{attribute addProperty BoxType "EK1122-0000-0018"}
{attribute addProperty Id "A_0060_AT2020_0250_0019_AT2020_0250A_0060_AT2020_0250_0019_AT2020_0250_D1D8CBA264080Beckhoff_AT2xxxsub_EK1100EK1100_179A0949162A_0001_AT2000_0233_0022AT2000_050BA88864080A_0002_AT2000_0233_0023AT2000_050BA88864080A_0003_AT2000_0233_0024AT2000_050BA88864080A_0004_AT2000_0250_0016AT2000_9506A48267284A_0005_AT2000_0250_0017AT2000_9506A48267284A_0006_AT2000_0250_0018AT2000_9506A48267284A_0007_AT2000_0250_0019AT2000_9506A48267284A_0008_AT2000_0250_0020AT2000_9506A48267284A_0009_AT2000_0250_0021AT2000_9506A48267284A_0010_AT2000_0250_0022AT2000_9506A48267284A_0011_AT2000_0250_0023AT2000_9506A48267284A_0012_AT2001_0250_0016AT2001_9506A48267284A_0013_AT2001_0250_0017AT2001_9506A48267284A_0014_AT2001_0250_0018AT2001_9506A48267284A_0015_AT2001_0250_0019AT2001_9506A48267284A_0016_AT2001_0250_0020AT2001_9506A48267284A_0017_AT2001_0250_0022AT2001_9506A48267284A_0018_AT2001_0250_0023AT2001_9506A48267284A_0019_AT2001_0250_0024AT2001_9506A48267284A_0020_AT2002_0249_0021AT2002_9506A48267284A_0021_AT2002_0249_0022AT2002_9506A48267284A_0022_AT2002_0249_0023AT2002_9506A48267284A_0023_AT2002_0250_0022AT2002_9506A48267284A_0024_AT2002_0250_0023AT2002_9506A48267284A_0025_AT2002_0250_0024AT2002_9506A48267284A_0026_AT2020_0250_0018AT2020_9506A48267284A_0027_AT2020_0250_0021AT2020_9506A48267284A_0028_AT2021_0250_0018AT2021_9506A48267284A_0029_AT2021_0250_0020AT2021_9506A48267284A_0030_AT2025_0250_0018AT2025_9506A48267284A_0031_AT2026_0250_0021AT2026_9506A48267284A_0032_AT2026_0250_0023AT2026_9506A48267284A_0033_AT2040_0250_0018AT2040_9506A48267284A_0034_AT2040_0250_0019AT2040_9506A48267284A_0035_AT2040_0250_0020AT2040_9506A48267284A_0036_AT2040_0250_0021A_0036_AT2040_0250_0021_02D2816B64080A_0037_AT2040_0250_0022A_0037_AT2040_0250_0022_F543FD7364080A_0038_AT2040_0250_0023A_0038_AT2040_0250_0023_F11EC84664080A_0039_AT2040_0250_0024A_0039_AT2040_0250_0024_E1E41A1064080A_0040_AT2041_0250_0018A_0040_AT2041_0250_0018_12B9905D64080A_0041_AT2041_0250_0019A_0041_AT2041_0250_0019_5F65D83164080A_0042_AT2041_0250_0020A_0042_AT2041_0250_0020_102CD79B64080A_0043_AT2041_0250_0021A_0043_AT2041_0250_0021_00D605CD64080A_0044_AT2041_0250_0022A_0044_AT2041_0250_0022_EDE0E1B464080A_0045_AT2041_0250_0023A_0045_AT2041_0250_0023_3AEB85C764080A_0046_AT2042_0250_0024A_0046_AT2042_0250_0024_1AE974B864080A_0047_AT2050_0500_0016A_0047_AT2050_0500_0016_ED7808A064080A_0048_AT2050_0500_0017A_0048_AT2050_0500_0017_6811D0ED64080A_0049_AT2050_0500_0018A_0049_AT2050_0500_0018_289538B264080A_0050_AT2050_0500_0019A_0050_AT2050_0500_0019_16FCA7F964080A_0051_AT2050_0500_0020A_0051_AT2050_0500_0020_887F94A764080A_0052_AT2050_0500_0021A_0052_AT2050_0500_0021_B6160BEC64080A_0053_AT2050_0500_0022A_0053_AT2050_0500_0022_1DEC9EBC64080A_0054_AT2050_0500_0023A_0054_AT2050_0500_0023_99CF05DF64080A_0055_AT2050_0500_0024A_0055_AT2050_0500_0024_061BAB1564080A_0056_AT2050_0501_0017A_0056_AT2050_0501_0017_8372735864080A_0057_AT2050_0501_0020A_0057_AT2050_0501_0020_74E30F4064080A_0058_AT2050_0501_0021A_0058_AT2050_0501_0021_C12219F464080A_0061_AT2020_0250_0023_AT2020_0250A_0061_AT2020_0250_0023_AT2020_0250_98D9E94964080A_0062_AT2025_0250_0020_AT2025_0250A_0062_AT2025_0250_0020_AT2025_0250_D505A12564080A_0063_AT2025_0250_0022_AT2025_0250A_0063_AT2025_0250_0022_AT2025_0250_FB2CCE7664080A_0064_AT2025_0250_0023_AT2025_0250A_0064_AT2025_0250_0023_AT2025_0250_28C9970A64080A_0065_AT2026_0250_0019_AT2026_0250A_0065_AT2026_0250_0019_AT2026_0250_ADA04F4764080A_0066_AT2026_0250_0020_AT2026_0250A_0066_AT2026_0250_0020_AT2026_0250_5A31335F64080A_0067_AT2026_0250_0022_AT2026_0250A_0067_AT2026_0250_0022_AT2026_0250_D8AB0CE364080A_0068_AT2026_0250_0024_AT2026_0250A_0068_AT2026_0250_0024_AT2026_0250_C0DF91BF64080A_0069_AT2050_0501_0019_AT2050_0501A_0069_AT2050_0501_0019_AT2050_0501_33653EE264080A_0070_AT2050_0501_0022_AT2050_0501A_0070_AT2050_0501_0022_AT2050_0501_239FECB464080A_0071_AT2050_0501_0023_AT2050_0501A_0071_AT2050_0501_0023_AT2050_0501_196D5B8364080A_0072_AT2050_0501_0024_AT2050_0501A_0072_AT2050_0501_0024_AT2050_0501_54B113EF64080"}
{attribute addProperty CRC "2763086114"}
{attribute addProperty SizeInBites "46480"}
{attribute addProperty SizeInBytes "5810"}
TYPE Beckhoff_AT2xxxEK1122_A4B15922 EXTENDS EK1122_179A0949 :
STRUCT
	{attribute addProperty Name "A_0060_AT2020_0250_0019_AT2020_0250"}
	A_0060_AT2020_0250_0019_AT2020_0250 : A_0060_AT2020_0250_0019_AT2020_0250_D1D8CBA2;
	{attribute addProperty Name "Beckhoff_AT2xxxsub_EK1100"}
	Beckhoff_AT2xxxsub_EK1100 : EK1100_179A0949;
	{attribute addProperty Name "A_0001_AT2000_0233_0022"}
	A_0001_AT2000_0233_0022 : AT2000_050BA888;
	{attribute addProperty Name "A_0002_AT2000_0233_0023"}
	A_0002_AT2000_0233_0023 : AT2000_050BA888;
	{attribute addProperty Name "A_0003_AT2000_0233_0024"}
	A_0003_AT2000_0233_0024 : AT2000_050BA888;
	{attribute addProperty Name "A_0004_AT2000_0250_0016"}
	A_0004_AT2000_0250_0016 : AT2000_9506A482;
	{attribute addProperty Name "A_0005_AT2000_0250_0017"}
	A_0005_AT2000_0250_0017 : AT2000_9506A482;
	{attribute addProperty Name "A_0006_AT2000_0250_0018"}
	A_0006_AT2000_0250_0018 : AT2000_9506A482;
	{attribute addProperty Name "A_0007_AT2000_0250_0019"}
	A_0007_AT2000_0250_0019 : AT2000_9506A482;
	{attribute addProperty Name "A_0008_AT2000_0250_0020"}
	A_0008_AT2000_0250_0020 : AT2000_9506A482;
	{attribute addProperty Name "A_0009_AT2000_0250_0021"}
	A_0009_AT2000_0250_0021 : AT2000_9506A482;
	{attribute addProperty Name "A_0010_AT2000_0250_0022"}
	A_0010_AT2000_0250_0022 : AT2000_9506A482;
	{attribute addProperty Name "A_0011_AT2000_0250_0023"}
	A_0011_AT2000_0250_0023 : AT2000_9506A482;
	{attribute addProperty Name "A_0012_AT2001_0250_0016"}
	A_0012_AT2001_0250_0016 : AT2001_9506A482;
	{attribute addProperty Name "A_0013_AT2001_0250_0017"}
	A_0013_AT2001_0250_0017 : AT2001_9506A482;
	{attribute addProperty Name "A_0014_AT2001_0250_0018"}
	A_0014_AT2001_0250_0018 : AT2001_9506A482;
	{attribute addProperty Name "A_0015_AT2001_0250_0019"}
	A_0015_AT2001_0250_0019 : AT2001_9506A482;
	{attribute addProperty Name "A_0016_AT2001_0250_0020"}
	A_0016_AT2001_0250_0020 : AT2001_9506A482;
	{attribute addProperty Name "A_0017_AT2001_0250_0022"}
	A_0017_AT2001_0250_0022 : AT2001_9506A482;
	{attribute addProperty Name "A_0018_AT2001_0250_0023"}
	A_0018_AT2001_0250_0023 : AT2001_9506A482;
	{attribute addProperty Name "A_0019_AT2001_0250_0024"}
	A_0019_AT2001_0250_0024 : AT2001_9506A482;
	{attribute addProperty Name "A_0020_AT2002_0249_0021"}
	A_0020_AT2002_0249_0021 : AT2002_9506A482;
	{attribute addProperty Name "A_0021_AT2002_0249_0022"}
	A_0021_AT2002_0249_0022 : AT2002_9506A482;
	{attribute addProperty Name "A_0022_AT2002_0249_0023"}
	A_0022_AT2002_0249_0023 : AT2002_9506A482;
	{attribute addProperty Name "A_0023_AT2002_0250_0022"}
	A_0023_AT2002_0250_0022 : AT2002_9506A482;
	{attribute addProperty Name "A_0024_AT2002_0250_0023"}
	A_0024_AT2002_0250_0023 : AT2002_9506A482;
	{attribute addProperty Name "A_0025_AT2002_0250_0024"}
	A_0025_AT2002_0250_0024 : AT2002_9506A482;
	{attribute addProperty Name "A_0026_AT2020_0250_0018"}
	A_0026_AT2020_0250_0018 : AT2020_9506A482;
	{attribute addProperty Name "A_0027_AT2020_0250_0021"}
	A_0027_AT2020_0250_0021 : AT2020_9506A482;
	{attribute addProperty Name "A_0028_AT2021_0250_0018"}
	A_0028_AT2021_0250_0018 : AT2021_9506A482;
	{attribute addProperty Name "A_0029_AT2021_0250_0020"}
	A_0029_AT2021_0250_0020 : AT2021_9506A482;
	{attribute addProperty Name "A_0030_AT2025_0250_0018"}
	A_0030_AT2025_0250_0018 : AT2025_9506A482;
	{attribute addProperty Name "A_0031_AT2026_0250_0021"}
	A_0031_AT2026_0250_0021 : AT2026_9506A482;
	{attribute addProperty Name "A_0032_AT2026_0250_0023"}
	A_0032_AT2026_0250_0023 : AT2026_9506A482;
	{attribute addProperty Name "A_0033_AT2040_0250_0018"}
	A_0033_AT2040_0250_0018 : AT2040_9506A482;
	{attribute addProperty Name "A_0034_AT2040_0250_0019"}
	A_0034_AT2040_0250_0019 : AT2040_9506A482;
	{attribute addProperty Name "A_0035_AT2040_0250_0020"}
	A_0035_AT2040_0250_0020 : AT2040_9506A482;
	{attribute addProperty Name "A_0036_AT2040_0250_0021"}
	A_0036_AT2040_0250_0021 : A_0036_AT2040_0250_0021_02D2816B;
	{attribute addProperty Name "A_0037_AT2040_0250_0022"}
	A_0037_AT2040_0250_0022 : A_0037_AT2040_0250_0022_F543FD73;
	{attribute addProperty Name "A_0038_AT2040_0250_0023"}
	A_0038_AT2040_0250_0023 : A_0038_AT2040_0250_0023_F11EC846;
	{attribute addProperty Name "A_0039_AT2040_0250_0024"}
	A_0039_AT2040_0250_0024 : A_0039_AT2040_0250_0024_E1E41A10;
	{attribute addProperty Name "A_0040_AT2041_0250_0018"}
	A_0040_AT2041_0250_0018 : A_0040_AT2041_0250_0018_12B9905D;
	{attribute addProperty Name "A_0041_AT2041_0250_0019"}
	A_0041_AT2041_0250_0019 : A_0041_AT2041_0250_0019_5F65D831;
	{attribute addProperty Name "A_0042_AT2041_0250_0020"}
	A_0042_AT2041_0250_0020 : A_0042_AT2041_0250_0020_102CD79B;
	{attribute addProperty Name "A_0043_AT2041_0250_0021"}
	A_0043_AT2041_0250_0021 : A_0043_AT2041_0250_0021_00D605CD;
	{attribute addProperty Name "A_0044_AT2041_0250_0022"}
	A_0044_AT2041_0250_0022 : A_0044_AT2041_0250_0022_EDE0E1B4;
	{attribute addProperty Name "A_0045_AT2041_0250_0023"}
	A_0045_AT2041_0250_0023 : A_0045_AT2041_0250_0023_3AEB85C7;
	{attribute addProperty Name "A_0046_AT2042_0250_0024"}
	A_0046_AT2042_0250_0024 : A_0046_AT2042_0250_0024_1AE974B8;
	{attribute addProperty Name "A_0047_AT2050_0500_0016"}
	A_0047_AT2050_0500_0016 : A_0047_AT2050_0500_0016_ED7808A0;
	{attribute addProperty Name "A_0048_AT2050_0500_0017"}
	A_0048_AT2050_0500_0017 : A_0048_AT2050_0500_0017_6811D0ED;
	{attribute addProperty Name "A_0049_AT2050_0500_0018"}
	A_0049_AT2050_0500_0018 : A_0049_AT2050_0500_0018_289538B2;
	{attribute addProperty Name "A_0050_AT2050_0500_0019"}
	A_0050_AT2050_0500_0019 : A_0050_AT2050_0500_0019_16FCA7F9;
	{attribute addProperty Name "A_0051_AT2050_0500_0020"}
	A_0051_AT2050_0500_0020 : A_0051_AT2050_0500_0020_887F94A7;
	{attribute addProperty Name "A_0052_AT2050_0500_0021"}
	A_0052_AT2050_0500_0021 : A_0052_AT2050_0500_0021_B6160BEC;
	{attribute addProperty Name "A_0053_AT2050_0500_0022"}
	A_0053_AT2050_0500_0022 : A_0053_AT2050_0500_0022_1DEC9EBC;
	{attribute addProperty Name "A_0054_AT2050_0500_0023"}
	A_0054_AT2050_0500_0023 : A_0054_AT2050_0500_0023_99CF05DF;
	{attribute addProperty Name "A_0055_AT2050_0500_0024"}
	A_0055_AT2050_0500_0024 : A_0055_AT2050_0500_0024_061BAB15;
	{attribute addProperty Name "A_0056_AT2050_0501_0017"}
	A_0056_AT2050_0501_0017 : A_0056_AT2050_0501_0017_83727358;
	{attribute addProperty Name "A_0057_AT2050_0501_0020"}
	A_0057_AT2050_0501_0020 : A_0057_AT2050_0501_0020_74E30F40;
	{attribute addProperty Name "A_0058_AT2050_0501_0021"}
	A_0058_AT2050_0501_0021 : A_0058_AT2050_0501_0021_C12219F4;
	{attribute addProperty Name "A_0061_AT2020_0250_0023_AT2020_0250"}
	A_0061_AT2020_0250_0023_AT2020_0250 : A_0061_AT2020_0250_0023_AT2020_0250_98D9E949;
	{attribute addProperty Name "A_0062_AT2025_0250_0020_AT2025_0250"}
	A_0062_AT2025_0250_0020_AT2025_0250 : A_0062_AT2025_0250_0020_AT2025_0250_D505A125;
	{attribute addProperty Name "A_0063_AT2025_0250_0022_AT2025_0250"}
	A_0063_AT2025_0250_0022_AT2025_0250 : A_0063_AT2025_0250_0022_AT2025_0250_FB2CCE76;
	{attribute addProperty Name "A_0064_AT2025_0250_0023_AT2025_0250"}
	A_0064_AT2025_0250_0023_AT2025_0250 : A_0064_AT2025_0250_0023_AT2025_0250_28C9970A;
	{attribute addProperty Name "A_0065_AT2026_0250_0019_AT2026_0250"}
	A_0065_AT2026_0250_0019_AT2026_0250 : A_0065_AT2026_0250_0019_AT2026_0250_ADA04F47;
	{attribute addProperty Name "A_0066_AT2026_0250_0020_AT2026_0250"}
	A_0066_AT2026_0250_0020_AT2026_0250 : A_0066_AT2026_0250_0020_AT2026_0250_5A31335F;
	{attribute addProperty Name "A_0067_AT2026_0250_0022_AT2026_0250"}
	A_0067_AT2026_0250_0022_AT2026_0250 : A_0067_AT2026_0250_0022_AT2026_0250_D8AB0CE3;
	{attribute addProperty Name "A_0068_AT2026_0250_0024_AT2026_0250"}
	A_0068_AT2026_0250_0024_AT2026_0250 : A_0068_AT2026_0250_0024_AT2026_0250_C0DF91BF;
	{attribute addProperty Name "A_0069_AT2050_0501_0019_AT2050_0501"}
	A_0069_AT2050_0501_0019_AT2050_0501 : A_0069_AT2050_0501_0019_AT2050_0501_33653EE2;
	{attribute addProperty Name "A_0070_AT2050_0501_0022_AT2050_0501"}
	A_0070_AT2050_0501_0022_AT2050_0501 : A_0070_AT2050_0501_0022_AT2050_0501_239FECB4;
	{attribute addProperty Name "A_0071_AT2050_0501_0023_AT2050_0501"}
	A_0071_AT2050_0501_0023_AT2050_0501 : A_0071_AT2050_0501_0023_AT2050_0501_196D5B83;
	{attribute addProperty Name "A_0072_AT2050_0501_0024_AT2050_0501"}
	A_0072_AT2050_0501_0024_AT2050_0501 : A_0072_AT2050_0501_0024_AT2050_0501_54B113EF;
END_STRUCT
END_TYPE

(* stored: Version 1.2.0.0, ProductVersion 3.1.4024.9
   DUT Beckhoff_AT2xxxEK1122_A4B15922: Id {23e6654c-bc76-42fc-b04e-f1fe8f7c559f} *)
